PROGRAM MAIN
VAR
	bProjectB : BOOL;
	fbLogger : FB_LogHandler;
END_VAR

fbLogger();

END_PROGRAM

(* stored: Version 1.1.0.1, ProductVersion 3.1.4022.18
   POU MAIN: Id {6938e8df-3947-445a-b470-1bf73db87944}, SpecialFunc None *)
